(* CoDeSys 2.3.9.41 project: плк100_икз.pro *)
(* Libraries: Util.lib 1.6.07 09:40:58, UNM.lib 14.2.06 11:27:08, STANDARD.LIB 20.2.06 12:31:06, IECSFC.LIB 20.2.06 12:31:00, SYSLIBTIME.LIB 20.2.06 12:31:16, SYSTASKINFO.LIB 20.2.06 12:31:38, ANALYZATION.LIB 20.2.06 12:30:58, SYSLIBCALLBACK.LIB 20.2.06 12:31:08, oscat_basic_333.lib 17.7.18 22:33:05 *)

(* PLC configuration (modules and I/O channels)
AT %IB0.0 [ByteInput] 8 discrete inputs
DO0 AT %QX1.0 [BitOutput] relay
DO1 AT %QX2.0 [BitOutput] relay
DO2 AT %QX3.0 [BitOutput] relay
Discrete output - relay [ID102] node 4, in %IB4 out %QB4 {PinCount = 1; SafeValueBool = FALSE; Visibility = No}
  AT %QX4.0 [BitOutput] relay
Discrete output - relay [ID102] node 5, in %IB5 out %QB5 {PinCount = 1; SafeValueBool = FALSE; Visibility = No}
  AT %QX5.0 [BitOutput] relay
Discrete output - relay [ID102] node 6, in %IB6 out %QB6 {PinCount = 1; SafeValueBool = FALSE; Visibility = No}
  AT %QX6.0 [BitOutput] relay
AT %QX7.0 [BitOutput] Special output
TCP [TCP_ID221] node 0, in %IB8.0.0 out %QB8.0.0 {RemotePort = 502; Visibility = No}
AT %QB8.1.0 [ByteOutput]
AT %QB8.2.0 [ByteOutput]
*)

(* POU PLC_PRG, ST *)
PROGRAM PLC_PRG
VAR
	out8:BYTE:=1;
	out9:BYTE:=1;
	timer8: TON;
	timer9: TON;
	flag8:BOOL:=FALSE;

	flag9:BOOL:=FALSE;
END_VAR
(*дискретные входы пересылаем в модбас*)
(*
output0:=input0;
output1:=input1;
output2:=input2;
output3:=input3;
output4:=input4;
output5:=input5;
output6:=input6;
output7:=input7;
*)

IF(input0>0) THEN
	output0:=1;
END_IF;

IF(input1>0) THEN
	output1:=1;
END_IF;

IF(input2>0) THEN
	output2:=1;
END_IF;

IF(input3>0) THEN
	output3:=1;
END_IF;

IF(input4>0) THEN
	output4:=1;
END_IF;

IF(input5>0) THEN
	output5:=1;
END_IF;


IF(input6>0) THEN
	output6:=1;
END_IF;

IF(input7>0) THEN
	output7:=1;
END_IF;




(*управление выходом по модбасу*)

IF(output8>0) THEN
	flag8:=TRUE;
	output0:=0;
	output1:=0;
	output2:=0;
	output3:=0;
	output4:=0;
	output5:=0;
	output6:=0;
	output7:=0;
	output8:=0;
END_IF

timer8(IN := flag8, PT := T#2s);
IF timer8.Q THEN
	flag8:=FALSE;
END_IF;


IF (flag8) THEN
	DO0:=1;
ELSE
	DO0:=0;
END_IF;


IF(output9>0) THEN
	flag9:=TRUE;
	output9:=0;
END_IF

timer9(IN := flag9, PT := T#2s);
IF timer9.Q THEN
	flag9:=FALSE;
END_IF;


IF (flag9) THEN
	DO1:=1;
ELSE
	DO1:=0;
END_IF;
END_PROGRAM
